// TIA Portal V19 export
FUNCTION_BLOCK "LEXCHANGETRAY_Pcacuator"   // FB153, LAD
TITLE = PCAcuator
AUTHOR : SUP/zhang shi long
FAMILY : SUP
// get pc information
// stored: Access Published, MemoryReserve 100, SetENOAutomatically false
   VAR_IN_OUT
      controlNode : "LEXCHANGETRAY_typePc_controlNode";
      hmiInterface : "LEXCHANGETRAY_typePc_Interface";
   END_VAR
   VAR
      instrandomNgGenerator : "LEXCHANGETRAY_RandomNgInterface";
      statSimProcessMonitor { ExternalAccessible := 'False'; ExternalVisible := 'False'; ExternalWritable := 'False'} : "LEXCHANGETRAY_typePc_Monitor";
   END_VAR
BEGIN

REGION Network 1: DESCRIPTION
END_REGION

REGION Network 2: INITIALISATION
END_REGION

REGION Network 3: PROGRAM LOGIC
END_REGION

REGION Network 4
   // cellsResult : TRUE OK FALSE NG
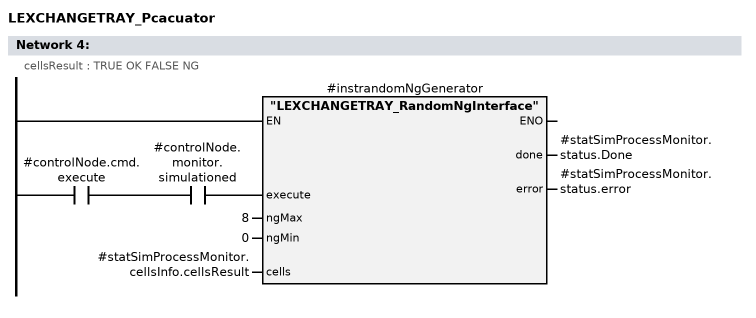
   RUNG wire#powerrail
      #instrandomNgGenerator(execute := wire#w1, ngMax := 8, ngMin := 0, cells := #statSimProcessMonitor.cellsInfo.cellsResult, done => #statSimProcessMonitor.status.Done, error => #statSimProcessMonitor.status.error)
   END_RUNG
   RUNG wire#powerrail
      Contact( #controlNode.cmd.execute )
      Contact( #controlNode.monitor.simulationed )
   END_RUNG wire#w1
   // the same network as SCL:
   #instrandomNgGenerator(execute := #controlNode.cmd.execute AND #controlNode.monitor.simulationed,   // "LEXCHANGETRAY_RandomNgInterface"
                          ngMax := 8,
                          ngMin := 0,
                          cells := #statSimProcessMonitor.cellsInfo.cellsResult,
                          done => #statSimProcessMonitor.status.Done,
                          error => #statSimProcessMonitor.status.error);
END_REGION

REGION Network 5: OUTPUTS
END_REGION

REGION Network 6 (SCL)
   IF #controlNode.cmd.raiseError THEN
       // Statement section IF

       #statSimProcessMonitor.status.error:=TRUE;
   END_IF;
   IF #controlNode.cmd.resetError THEN
       #controlNode.cmd.resetError:=

       #statSimProcessMonitor.status.error := FALSE;
   END_IF;
END_REGION

REGION Network 7 (SCL)
   IF #controlNode.monitor.simulationed THEN
       #statSimProcessMonitor.cellsInfo.cellSize := 24;

   END_IF;
END_REGION

REGION Network 10 (SCL)
   #statSimProcessMonitor.simulationed:=
   #hmiInterface.monitor.simulationed :=
   #controlNode.monitor.simulationed := #controlNode.cmd.simActive;
   IF #controlNode.monitor.simulationed THEN

       #hmiInterface.monitor:=#controlNode.monitor:=#statSimProcessMonitor;
   ELSE
       #hmiInterface.monitor := #controlNode.monitor := #statSimProcessMonitor;

   END_IF;
END_REGION
END_FUNCTION_BLOCK
